TYPE HMIRFIDInterface :
STRUCT
	RFIDStatus	:	HMIRFIDStatusInterface;
	RFIDControl	:	HMIRFIDControlInterface;
	RFIDData	:	HMIRFIDDataInterface;
END_STRUCT
END_TYPE

(* stored: Version 1.1.0.1
   DUT HMIRFIDInterface: Id {1b526505-33bd-42a4-a645-94e60f72605b} *)
